// Interlock logic for the Dump Chiller
FUNCTION F_DumpChillerEnable : BOOL
VAR_INPUT
END_VAR
VAR_IN_OUT CONSTANT
	stErrors : ST_ErrorStates; // Currently detected errors
END_VAR
VAR
END_VAR

F_DumpChillerEnable := FALSE;

// Disable dump chiller if there's a hardware failure
IF stErrors.bHardwareFailure THEN
	RETURN;
END_IF

// Disable dump chiller for these leak conditions
IF stErrors.bLeakOpticalTableAmphosOn OR stErrors.bLeakOpticalTableNoLaser OR stErrors.bLeakOpcpaCarbideOn OR stErrors.bLeakUnderTable THEN
	RETURN;
END_IF

F_DumpChillerEnable := TRUE;

END_FUNCTION

(* stored: Version 1.1.0.1, ProductVersion 3.1.4020.14
   POU F_DumpChillerEnable: Id {eacb95fa-49ef-4c8d-8057-f0d541675cea}, SpecialFunc None *)
